// TIA Portal V19 export
FUNCTION "BA_WXL" : Void   // FC4, STL
{ S7_Optimized_Access := 'FALSE' }
AUTHOR : MS
// stored: AutoNumber false
   VAR_TEMP
      Evnt_Nbr : Byte;
   END_VAR
   VAR CONSTANT
      Not_Halt : USInt;
      Tipp : USInt := 1;
      Hand : USInt := 2;
      Automat_Aus : USInt := 3;
      Automat_Ein : USInt := 4;
   END_VAR
BEGIN

NETWORK
TITLE = Not-Aus ist betätigt
      A     "DB_ANLAGE".config.Anl_getaktet;
      =     "DB_Panel_OVERVIEW".SPS_getaktet;

      A     "DB_ANLAGE".IN.S_Not_Aus;
      JC    off;

//Automatikbetrieb
      A     "DB_ANLAGE".BA.Not_Aus;
      R     "DB_ANLAGE".BA.Not_Aus;
      R     "DB_ANLAGE".BA.Tippbetrieb;
      R     "DB_ANLAGE".BA.Handbetrieb;
      R     "DB_ANLAGE".BA.Automat_ein;
      S     "DB_ANLAGE".BA.Automat_aus;

      A     "DB_ANLAGE".IN.Automat_ein;
      FP    "DB_ANLAGE".BA.FP_Automat_ein;
      R     "DB_ANLAGE".BA.Not_Aus;
      R     "DB_ANLAGE".BA.Tippbetrieb;
      R     "DB_ANLAGE".BA.Handbetrieb;
      S     "DB_ANLAGE".BA.Automat_ein;
      R     "DB_ANLAGE".BA.Automat_aus;

      A     "DB_ANLAGE".IN.Automat_aus;
      R     "DB_ANLAGE".BA.Not_Aus;
      R     "DB_ANLAGE".BA.Tippbetrieb;
      R     "DB_ANLAGE".BA.Handbetrieb;
      R     "DB_ANLAGE".BA.Automat_ein;
      S     "DB_ANLAGE".BA.Automat_aus;

      A     "DB_ANLAGE".BA.Automat_ein;
      O     "DI_FW_MANAGER".Auto.Anlage;
      O     "DB_ANLAGE".IN.Lamp_Test;
      =     "DB_ANLAGE".OUT.MD_Auto;

//Handbetrieb
      A     "DB_ANLAGE".IN.BA_Hand;
      R     "DB_ANLAGE".BA.Not_Aus;
      R     "DB_ANLAGE".BA.Tippbetrieb;
      S     "DB_ANLAGE".BA.Handbetrieb;
      R     "DB_ANLAGE".BA.Automat_ein;
      R     "DB_ANLAGE".BA.Automat_aus;

//Einrichten
      A     "DB_ANLAGE".IN.BA_Tipp;
      R     "DB_ANLAGE".BA.Not_Aus;
      S     "DB_ANLAGE".BA.Tippbetrieb;
      R     "DB_ANLAGE".BA.Handbetrieb;
      R     "DB_ANLAGE".BA.Automat_ein;
      R     "DB_ANLAGE".BA.Automat_aus;

//Auto-Stop
      A     "DB_ANLAGE".BA.Automat_aus;
      R     "DB_ANLAGE".BA.Not_Aus;
      R     "DB_ANLAGE".BA.Tippbetrieb;
      R     "DB_ANLAGE".BA.Handbetrieb;
      R     "DB_ANLAGE".BA.Automat_ein;

      L     #Automat_Ein;
      A     "DB_ANLAGE".BA.Automat_ein;
      JC    A_BA;
      L     #Automat_Aus;
      A     "DB_ANLAGE".BA.Automat_aus;
      JC    A_BA;
      L     #Hand;
      A     "DB_ANLAGE".BA.Handbetrieb;
      JC    A_BA;
      L     #Tipp;
      A     "DB_ANLAGE".BA.Tippbetrieb;
      JC    A_BA;
      L     #Not_Halt;
A_BA: T     "Panel".Betriebsart.Anzeige;
      JU    ende;

//alles aus
off:  R     "DB_ANLAGE".BA.free0;
      R     "DB_ANLAGE".BA.free1;
      R     "DB_ANLAGE".BA.Tippbetrieb;
      R     "DB_ANLAGE".BA.Handbetrieb;
      R     "DB_ANLAGE".BA.Automat_ein;
      R     "DB_ANLAGE".BA.Automat_aus;
      S     "DB_ANLAGE".BA.Not_Aus;
      L     #Not_Halt;
      T     "Panel".Betriebsart.Anzeige;

ende: OPN   "DB_ANLAGE";
      L     %DBW0;  //Betriebsart SPS
      OPN   "DB_Panel_OVERVIEW";
      T     %DBW0;  //Betriebsart Visualisierung
      BE;
END_FUNCTION
